TYPE ModbusDint :
UNION
	rawdata		: ARRAY[0..1] OF WORD;
	value	: DINT;
END_UNION
END_TYPE

(* stored: Version 1.1.0.1
   DUT ModbusDint: Id {c679fe4b-1b45-47ee-b4f0-7a2b80938d6f} *)
